# B&R Automation Studio project ASCommon
Automation Studio 6.5.0.306; technology packages: mappCockpit 6.6.0, mappMotion 6.6.1, mappSafety 6.4.1, mappServices 6.6.0, mappView 6.6.0, OpcUaCs 6.6.0

## Configuration X20CP1686X

CPU 5APC4100.TGL1-000, AutomationRuntime 6.5.1, Build 11.3.0, Vc 6.5.0

### Task classes (Cpu.sw)
```
Cyclic#1:
  MoveAxis <- Motion.MoveAxis.prg
  SimConnect <- SimConnect.prg
  BoxCreate <- BoxLift.BoxCreate.BoxCreate.prg [disabled]
  InfeedUp <- BoxLift.InfeedUp.InfeedUp.prg [disabled]
  InfeedLow <- BoxLift.InfeedLow.InfeedLow.prg [disabled]
  Lift <- BoxLift.Lift.Lift.prg [disabled]
  Unload <- BoxLift.Unload.Unload.prg [disabled]
  MachineMan <- BoxLift.MachineManager.MachineManager.prg [disabled]
  MachineMa1 <- BoxLiftOOP.MachineManager.prg
Cyclic#4:
  LampTest <- LampTest.prg
  RecipeMan <- Recipe.RecipeMan.prg
  SafetyCtrl <- Safety.SafetyCtrl.prg
DataObjects: McAcpSys
NcDataObjects: McDriveLog
Binaries: McAcpDrv, udbdef, McAcpSim, mvLoader, TCLang, TCData, FWRules, ArSvcReg, mvConfig, BRRole, sysconf, iomap, asfw, ashwac, UaCsConfig, Config_2, Config_1, ashwd, arconfig, Role, WebServ, User, TC, OpcUaCfg
Libraries: runtime, sys_lib, FileIO, AsZip, McBase, MpBase, MpAxis, McAcpAx, McAxis, SfDomain, MpCom, MpRecipe, CoTrace, AsTCP, AsIecCon, AsIODiag, UaCoal, SfDomVis, astime, standard, AsEPL, AsIOAcc, SfDomDrv, AsUSB, MpSfDomMgr, UaCoalPrv, ArUser, ArSsl, powerlnk, UaCore, AsIoTrc
```

### Hardware
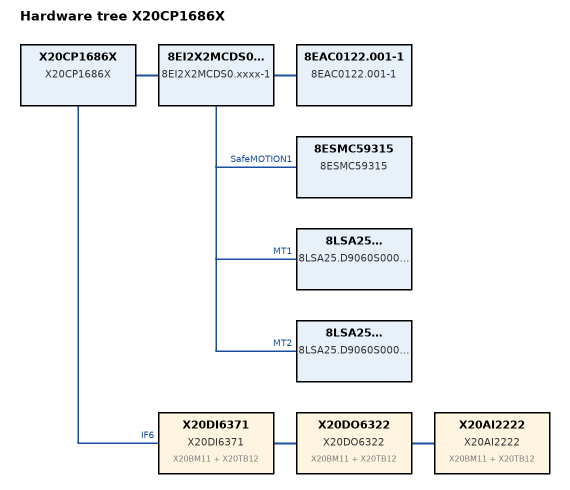
```
8EAC0122.001-1 : 8EAC0122.001-1 v3.0.0.0  [SS -> 8EI2X2MCDS0.xxxx-1.SS1]
  PlugInType = Encoder
  McAcoposTypeID = AcoposP3PlugInSConfig
  InterfaceType = Resolver
8EI2X2MCDS0.xxxx-1 : 8EI2X2MCDS0.xxxx-1 v2.4.0.3 (NodeNumber=1)  [PLK1 -> X20CP1686X.IF3 [Cable Type=PowerlinkCable, Length=10, Version=1.0.0.3]; MT2 -> 8LSA25.D9060S000-3a.MT]
  DriveConfiguration/Module:
    McAcoposTypeID = AcoposP3DConfig
    ActivateACOPOSSimulationOnPLC = 0
    PowerSupply = AC
  DriveConfiguration/Encoder:
    SafeEncInterface = EnDat22_SafeMOTION
  DriveConfiguration/Encoder/EncoderX41:
    InterfaceType = EnDatSafeMotion
  DriveConfiguration/Encoder/EncoderX42:
    InterfaceType = EnDatSafeMotion
  DriveConfiguration/Channel[1]/RealAxis:
    AxisReference = gAxis01
    MechanicalElementsIsInvisible = 0
  DriveConfiguration/Channel[1]/RealAxis/MechanicalElements/Gearbox:
    InputIsReadOnly = 0
    Input = 1
    OutputIsReadOnly = 0
    Output = 1
  DriveConfiguration/Channel[1]/RealAxis/MechanicalElements/RotaryToLinearTransformation:
    ReferenceDistanceIsReadOnly = 0
    ReferenceDistance = 1
  DriveConfiguration/Channel[1]/RealAxis:
    EncoderLink = OneEncoder
  DriveConfiguration/Channel[1]/RealAxis/Controller:
    ModeIsReadOnly = 0
    Mode = PositionController
  DriveConfiguration/Channel[1]/RealAxis/Homing:
    ModeIsReadOnly = 0
    Mode = Direct
    RestorePositionVariable = 
  DriveConfiguration/Channel[1]/RealAxis/StopReaction:
    QuickstopIsReadOnly = 0
    Quickstop = DecelerationLimit
    DriveErrorIsReadOnly = 0
    DriveError = DecelerationLimit
  DriveConfiguration/Channel[1]/RealAxis/MovementErrorLimits:
    PositionError = 10.0
    VelocityErrorMonitoring = Automatic1
  DriveConfiguration/Channel[1]/RealAxis:
    JerkFilterIsReadOnly = 0
    JerkFilter = NotUsed
    ZeroVibrationFilter = NotUsed
  DriveConfiguration/Channel[1]/RealAxis/DigitalInputs/HomingSwitch:
    SourceIsReadOnly = 0
    Source = NotUsed
    Level = High
  DriveConfiguration/Channel[1]/RealAxis/DigitalInputs/PositiveLimitSwitch:
    SourceIsReadOnly = 0
    Source = NotUsed
    Level = High
  DriveConfiguration/Channel[1]/RealAxis/DigitalInputs/NegativeLimitSwitch:
    SourceIsReadOnly = 0
    Source = NotUsed
    Level = High
  DriveConfiguration/Channel[1]/RealAxis/DigitalInputs/Trigger1:
    Source = X8Trigger1
    Level = High
  DriveConfiguration/Channel[1]/RealAxis/DigitalInputs/Trigger2:
    Source = X8Trigger2
    Level = High
  DriveConfiguration/Channel[1]/RealAxis/DigitalInputs/Quickstop:
    Input = Trigger2
  DriveConfiguration/Channel[1]/RealAxis/Simulation:
    SimulationModeOnPLC = SetValueGeneration
    SimulationModeOnACOPOS = NotUsed
  DriveConfiguration/Channel[1]:
    VirtualAxis = NotUsed
    ExternalEncoderAxis = NotUsed
  DriveConfiguration/Channel[2]/RealAxis:
    AxisReference = 
    MechanicalElementsIsInvisible = 0
  DriveConfiguration/Channel[2]/RealAxis/MechanicalElements/Gearbox:
    InputIsReadOnly = 0
    Input = 1
    OutputIsReadOnly = 0
    Output = 1
  DriveConfiguration/Channel[2]/RealAxis/MechanicalElements/RotaryToLinearTransformation:
    ReferenceDistanceIsReadOnly = 0
    ReferenceDistance = 1
  DriveConfiguration/Channel[2]/RealAxis:
    EncoderLink = OneEncoder
  DriveConfiguration/Channel[2]/RealAxis/Controller:
    ModeIsReadOnly = 0
    Mode = PositionController
  DriveConfiguration/Channel[2]/RealAxis/Homing:
    ModeIsReadOnly = 0
    Mode = Direct
    RestorePositionVariable = 
  DriveConfiguration/Channel[2]/RealAxis/StopReaction:
    QuickstopIsReadOnly = 0
    Quickstop = DecelerationLimit
    DriveErrorIsReadOnly = 0
    DriveError = DecelerationLimit
  DriveConfiguration/Channel[2]/RealAxis/MovementErrorLimits:
    PositionError = 10.0
    VelocityErrorMonitoring = Automatic1
  DriveConfiguration/Channel[2]/RealAxis:
    JerkFilterIsReadOnly = 0
    JerkFilter = NotUsed
    ZeroVibrationFilter = NotUsed
  DriveConfiguration/Channel[2]/RealAxis/DigitalInputs/HomingSwitch:
    SourceIsReadOnly = 0
    Source = NotUsed
    Level = High
  DriveConfiguration/Channel[2]/RealAxis/DigitalInputs/PositiveLimitSwitch:
    SourceIsReadOnly = 0
    Source = NotUsed
    Level = High
  DriveConfiguration/Channel[2]/RealAxis/DigitalInputs/NegativeLimitSwitch:
    SourceIsReadOnly = 0
    Source = NotUsed
    Level = High
  DriveConfiguration/Channel[2]/RealAxis/DigitalInputs/Trigger1:
    Source = X8Trigger1
    Level = High
  DriveConfiguration/Channel[2]/RealAxis/DigitalInputs/Trigger2:
    Source = X8Trigger2
    Level = High
  DriveConfiguration/Channel[2]/RealAxis/DigitalInputs/Quickstop:
    Input = Trigger2
  DriveConfiguration/Channel[2]/RealAxis/Simulation:
    SimulationModeOnPLC = SetValueGeneration
    SimulationModeOnACOPOS = NotUsed
  DriveConfiguration/Channel[2]:
    VirtualAxis = NotUsed
    ExternalEncoderAxis = NotUsed
8ESMC59315 : 8ESMC59315 v2.4.0.0  [SafeMOTION -> 8EI2X2MCDS0.xxxx-1.SafeMOTION1]
8LSA25.D9060S000-3 : 8LSA25.D9060S000-3 v2.2.0.2  [MT -> 8EI2X2MCDS0.xxxx-1.MT1]
  M1/MotorParameters:
    MOTOR_AMB_TEMP_RATED = 40
  M1/MotorParameters/TemperatureSensor:
    MOTOR_TEMPSENS_LIM = 130
8LSA25.D9060S000-3a : 8LSA25.D9060S000-3 v2.2.0.2  [MT -> 8EI2X2MCDS0.xxxx-1.MT2]
  M1/MotorParameters:
    MOTOR_AMB_TEMP_RATED = 40
  M1/MotorParameters/TemperatureSensor:
    MOTOR_TEMPSENS_LIM = 130
X20AI2222 : X20AI2222 v1.4.0.0  [SS1 -> X20TB12b.SS; SL -> X20BM11b.SL1]
X20BM11 : X20BM11 v1.1.0.0  [X2X1 -> X20CP1686X.IF6]
X20BM11a : X20BM11 v1.1.0.0  [X2X1 -> X20BM11.X2X2]
X20BM11b : X20BM11 v1.1.0.0  [X2X1 -> X20BM11a.X2X2]
X20CP1686X : X20CP1686X v1.8.2.0
  Connector IF2:
    ActivateDevice = 1
    HostName = ascommon
    Mode = Manual
    InternetAddress = 192.168.0.10
    SubnetMask = 255.255.255.0
    ActivateSnmp = 2
  Connector IF3:
    EplHostName = ascommon
    HostName = ascommon
  ConfigurationID = ASCommon_X20CP1686X
  Simulation = 1
  EnableUsbRemoteInstall = 1
  FileDevice1
  FileDeviceName1 = USER
  FileDevicePath1 = USER_PATH
  TimeZone = 140
  ActivateDaylightSavingTime = 1
  ActivateSntp = 1
  SntpcServAddr1 = 10.43.10.23
  SntpcServAddr2 = 10.43.10.24
  EthernetHostName = ascommon
  ActivateWebServer = 1
  HttpsSslCfg = WebServConf
  ActivateSdm = 1
X20DI6371 : X20DI6371 v1.2.2.0  [SS1 -> X20TB12.SS; SL -> X20BM11.SL1]
X20DO6322 : X20DO6322 v1.4.1.0  [SS1 -> X20TB12a.SS; SL -> X20BM11a.SL1]
X20TB12 : X20TB12 v1.0.0.0
X20TB12a : X20TB12 v1.0.0.0
X20TB12b : X20TB12 v1.0.0.0
```

### IoMap.iom - X20CP1686X/IoMap.iom
```iecst
VAR_CONFIG
	::LampTest:diSwitch AT %IX."X20DI6371".DigitalInput01;
	::SafetyCtrl:di_Reset AT %IX."X20DI6371".DigitalInput03;
	::LampTest:doLamp AT %QX."X20DO6322".DigitalOutput01;
	::LampTest:doLamp AT %QX."X20DO6322".DigitalOutput02;
	::LampTest:doLamp AT %QX."X20DO6322".DigitalOutput03;
END_VAR
```

### PvMap.vvm - X20CP1686X/PvMap.vvm
```iecst
VAR_CONFIG
	::InfeedUp:IO.doInfeed1Conveyor AT %Q.::SimConnect:SimOutputs.doInfeed1Conveyor; (*Insert your comment here...*)
	::InfeedUp:IO.aoInfeed1ConveyorSetSpeed AT %Q.::SimConnect:SimOutputs.aoInfeed1ConveyorSetSpeed; (*Insert your comment here...*)
	::SimConnect:SimInputs.diInfeed1BoxDetection AT %Q.::InfeedUp:IO.diInfeed1BoxDetection; (*Insert your comment here...*)
	::InfeedLow:IO.doInfeed2Conveyor AT %Q.::SimConnect:SimOutputs.doInfeed2Conveyor; (*Insert your comment here...*)
	::InfeedLow:IO.aoInfeed2ConveyorSetSpeed AT %Q.::SimConnect:SimOutputs.aoInfeed2ConveyorSetSpeed; (*Insert your comment here...*)
	::SimConnect:SimInputs.diInfeed2BoxDetection AT %Q.::InfeedLow:IO.diInfeed2BoxDetection; (*Insert your comment here...*)
	::BoxCreate:IO.aoEntrance1ConveyorSetSpeed AT %Q.::SimConnect:SimOutputs.aoEntrance1ConveyorSetSpeed; (*Insert your comment here...*)
	::BoxCreate:IO.aoEntrance2ConveyorSetSpeed AT %Q.::SimConnect:SimOutputs.aoEntrance2ConveyorSetSpeed; (*Insert your comment here...*)
	::BoxCreate:IO.aoInfeed1BoxCreationInterval AT %Q.::SimConnect:SimOutputs.aoInfeed1BoxCreationInterval; (*Insert your comment here...*)
	::BoxCreate:IO.aoInfeed2BoxCreationInterval AT %Q.::SimConnect:SimOutputs.aoInfeed2BoxCreationInterval; (*Insert your comment here...*)
	::BoxCreate:IO.doStopBoxCreation AT %Q.::SimConnect:SimOutputs.doStopBoxCreation; (*Insert your comment here...*)
	::Lift:IO.doLiftUp AT %Q.::SimConnect:SimOutputs.doLiftUp; (*Insert your comment here...*)
	::Lift:IO.doLiftDown AT %Q.::SimConnect:SimOutputs.doLiftDown; (*Insert your comment here...*)
	::Lift:IO.doLiftConveyor AT %Q.::SimConnect:SimOutputs.doLiftConveyor; (*Insert your comment here...*)
	::Lift:IO.aoLiftSetSpeed AT %Q.::SimConnect:SimOutputs.aoLiftSetSpeed; (*Insert your comment here...*)
	::Lift:IO.aoLiftConveyorSetSpeed AT %Q.::SimConnect:SimOutputs.aoLiftConveyorSetSpeed; (*Insert your comment here...*)
	::SimConnect:SimInputs.diLiftPositionInfeed1 AT %Q.::Lift:IO.diLiftPositionInfeed1; (*Insert your comment here...*)
	::SimConnect:SimInputs.diLiftPositionInfeed2 AT %Q.::Lift:IO.diLiftPositionInfeed2; (*Insert your comment here...*)
	::SimConnect:SimInputs.diLiftPositionUnload AT %Q.::Lift:IO.diLiftPositionUnload; (*Insert your comment here...*)
	::SimConnect:SimInputs.diLiftBoxDetection AT %Q.::Lift:IO.diLiftBoxDetection; (*Insert your comment here...*)
	::Unload:IO.aoUnloadConveyorSetSpeed AT %Q.::SimConnect:SimOutputs.aoUnloadConveyorSetSpeed; (*Insert your comment here...*)
	::SimConnect:SimInputs.diUnloadBoxDetection AT %Q.::Unload:IO.diUnloadBoxDetection; (*Insert your comment here...*)
END_VAR
```

### Config_1.axis - X20CP1686X/mappMotion/Config_1.axis
```
Element gAxis01 (Type=axis)
  BaseType = RotaryPeriodic
  MovementLimits = Internal
  Alarms = None
```

### Config_2.mprecipexml - X20CP1686X/mappServices/Config_2.mprecipexml
```
Element gRecipeXml (Type=mprecipexml)
  mapp.Gen:
    Enable = TRUE
    EnableCockpit = TRUE
    TaskClass = 4
    Audit = TRUE
    Parent
  mapp.Recipe.Xml:
    AutoSave = Standard
    Encryption = FALSE
    PassPhrase
    AutoExtension = TRUE
    Signature = Disabled
  Alarms = MpAlarmX
    mapp.AlarmX.Core.Configuration:
      [0]:
        Name = SaveFailed
        Message = {$BR/mapp/MpRecipeXml/Alarms/SaveFailed}
        Code = 0
        Severity = 1
        Behavior = EdgeAlarm
          AutoReset = TRUE
          Acknowledge = 1
          Confirm = 0
          MultipleInstances = TRUE
          ReactionWhilePending = TRUE
          Async = FALSE
          Recording:
            InactiveToActive = TRUE
            ActiveToInactive = FALSE
            UnacknowledgedToAcknowledged = TRUE
            UnconfirmedToConfirmed = TRUE
        Disable = FALSE
        AdditionalInformation1
        AdditionalInformation2
      [1]:
        Name = SaveFailedPartial
        Message = {$BR/mapp/MpRecipeXml/Alarms/SaveFailedPartial}
        Code = 0
        Severity = 1
        Behavior = EdgeAlarm
          AutoReset = TRUE
          Acknowledge = 1
          Confirm = 0
          MultipleInstances = TRUE
          ReactionWhilePending = TRUE
          Async = FALSE
          Recording:
            InactiveToActive = TRUE
            ActiveToInactive = FALSE
            UnacknowledgedToAcknowledged = TRUE
            UnconfirmedToConfirmed = TRUE
        Disable = FALSE
        AdditionalInformation1
        AdditionalInformation2
      [2]:
        Name = LoadFailed
        Message = {$BR/mapp/MpRecipeXml/Alarms/LoadFailed}
        Code = 0
        Severity = 1
        Behavior = EdgeAlarm
          AutoReset = TRUE
          Acknowledge = 1
          Confirm = 0
          MultipleInstances = TRUE
          ReactionWhilePending = TRUE
          Async = FALSE
          Recording:
            InactiveToActive = TRUE
            ActiveToInactive = FALSE
            UnacknowledgedToAcknowledged = TRUE
            UnconfirmedToConfirmed = TRUE
        Disable = FALSE
        AdditionalInformation1
        AdditionalInformation2
      [3]:
        Name = LoadFailedPartial
        Message = {$BR/mapp/MpRecipeXml/Alarms/LoadFailedPartial}
        Code = 0
        Severity = 1
        Behavior = EdgeAlarm
          AutoReset = TRUE
          Acknowledge = 1
          Confirm = 0
          MultipleInstances = TRUE
          ReactionWhilePending = TRUE
          Async = FALSE
          Recording:
            InactiveToActive = TRUE
            ActiveToInactive = FALSE
            UnacknowledgedToAcknowledged = TRUE
            UnconfirmedToConfirmed = TRUE
        Disable = FALSE
        AdditionalInformation1
        AdditionalInformation2
```

## Logical view

Binary libraries used (declarations not repeated): operator, runtime, astime, AsIecCon, brsystem, sys_lib, AsArSdm, AsZip, FileIO, standard, McBase 6.6.1, MpBase 6.6.0, MpAxis 6.6.1, McAcpAx 6.6.1, McAxis 6.6.1, SfDomain 6.4.1, MpCom 6.6.0, MpRecipe 6.6.0, CoTrace 6.6.0, MpAudit 6.6.0

### Password.txt
```
OPC UA Server:
	Nutzername: 	opcuauser
	Passwort:		.opcuauser

URL mappView Visu:
	http://127.0.0.1:81/index.html?visuId=mvStart
```

- Project.language (not shown)

### Global.var - Global variables
```iecst
VAR
	MpAxisParam : MpAxisBasicParType;
END_VAR
```


### Program Logical/Motion/MoveAxis (ANSIC)

#### Variables.var
```iecst
VAR
	Para : MpAxisBasicParType;
	mpAxisBasic_0 : MpAxisBasic;
END_VAR
```

#### compile_flags.txt
```
# This file is auto-generated by ASX. Do not edit manually, as changes may be overwritten.
# If you need to manually edit this file and prevent automatic updates, add "# MANUAL EDIT" to the first line.
-I
c:\projects_63\sps\Logical\Motion\MoveAxis
-I
c:\projects_63\sps\Temp\Includes\Motion\MoveAxis
-I
C:\Program Files (x86)\BrAutomation\AS6\AS\gnuinst\V11.3.0\6.0\i686-elf\include\c++\11.3.0
-I
C:\Program Files (x86)\BrAutomation\AS6\AS\gnuinst\V11.3.0\6.0\i686-elf\include\c++\11.3.0\i686-elf
-I
C:\Program Files (x86)\BrAutomation\AS6\AS\gnuinst\V11.3.0\6.0\i686-elf\include\c++\11.3.0\backward
-I
C:\Program Files (x86)\BrAutomation\AS6\AS\gnuinst\V11.3.0\6.0\lib\gcc\i686-elf\11.3.0\include
-I
C:\Program Files (x86)\BrAutomation\AS6\AS\gnuinst\V11.3.0\6.0\lib\gcc\i686-elf\11.3.0\include-fixed
-I
C:\Program Files (x86)\BrAutomation\AS6\AS\gnuinst\V11.3.0\6.0\i686-elf\include
-I
c:\projects_63\sps\Temp\Includes
-trigraphs
-fno-asm
-D
_DEFAULT_INCLUDES
-D
_SG4
--target=i686-elf
-fPIC
-Wall
```

#### Main.c
```c
#include <bur/plctypes.h>

#ifdef _DEFAULT_INCLUDES
	#include <AsDefault.h>
#endif

#define TRUE 1

void _INIT ProgramInit(void)
{
	mpAxisBasic_0.MpLink = &gAxis01;
	mpAxisBasic_0.Enable = TRUE;
	mpAxisBasic_0.Parameters = &Para;
}

void _CYCLIC ProgramCyclic(void)
{
	MpAxisBasic(&mpAxisBasic_0);
}

void _EXIT ProgramExit(void)
{

}
```

### Program Logical/Recipe/RecipeMan (IEC)

#### Cyclic.st - Cyclic code
```iecst
PROGRAM _INIT
	MpAxisParam := MpAxisParam;

	MpRecipeXml_0.Enable 	:= TRUE;
	MpRecipeXml_0.MpLink 	:= ADR(gRecipeXml);
	MpRecipeXml_0.DeviceName := ADR('Files');
	MpRecipeXml_0.FileName 	:= ADR(FileName);

	MpRecipeXml_0();

	MpRecipePar.Enable := TRUE;
	MpRecipePar.MpLink := ADR(gRecipeXml);
	MpRecipePar.PVName := ADR('MpAxisParam');

	MpRecipePar();

END_PROGRAM

PROGRAM _CYCLIC

	MpRecipeXml_0();
	MpRecipePar();

END_PROGRAM

PROGRAM _EXIT

	MpRecipeXml_0.Enable := FALSE;
	MpRecipeXml_0();

	MpRecipePar.Enable := FALSE;
	MpRecipePar();

END_PROGRAM
```

#### Variables.var - Local variables
```iecst
VAR
	MpRecipeXml_0 : MpRecipeXml;
	MpRecipePar : MpRecipeRegPar;
	FileName : {REDUND_UNREPLICABLE} STRING[80] := 'AxisParameter';
END_VAR
```

### Program Logical/Safety/SafetyCtrl (IEC)

#### Main.st - Init, cyclic, exit code
```iecst
PROGRAM _INIT

	MpAxisParam := MpAxisParam;
	gAxis01 	:= gAxis01;

END_PROGRAM

PROGRAM _CYCLIC

	di_Reset;

	diagCode_EStop;
	diagCode_LightCurtain;
	diagCode_Root;

END_PROGRAM

PROGRAM _EXIT

END_PROGRAM
```

#### Variables.var - Local variables
```iecst
VAR
	diagCode_EStop : UINT;
	diagCode_LightCurtain : UINT;
	diagCode_Root : UINT;
	di_Reset : BOOL;
END_VAR
```

### Package Logical/BoxLift - Project source code

### Package Logical/BoxLift/MachineManager - Automatic mode

### MachineManagerIF.typ - Module interface declaration (global visibility)
```iecst
TYPE
	AutomaticIFType : 	STRUCT  (*Communication interface for the Automatic module*)
		Cmd : AutomaticCmdType; (*Commands to the Automatic module*)
	END_STRUCT;
	AutomaticCmdType : 	STRUCT  (*Commands to the Automatic module*)
		Run : BOOL; (*Run the machine*)
	END_STRUCT;
END_TYPE
```

### MachineMangerIF.var - Module interface definition (global visibility)
```iecst
VAR
	gAutomatic : AutomaticIFType; (*Communication interface for the Automatic module*)
END_VAR
```

### Program Logical/BoxLift/MachineManager/MachineManager (IEC) - Automatic module functionality

#### Types.typ - Local data types
```iecst
(*Internal (private) data types*)

TYPE
	AutoStateEnum :
		(
		AUTO_IDLE,
		AUTO_WAIT_FOR_BOX,
		AUTO_PREPARE_UPPER_HANDOVER,
		AUTO_HANDOVER_UPPER_BOX,
		AUTO_PREPARE_LOWER_HANDOVER,
		AUTO_HANDOVER_LOWER_BOX,
		AUTO_HANDOVER_TO_UNLOAD,
		AUTO_UNLOAD_BOX
		);
END_TYPE
```

#### Variables.var - Local variables
```iecst
(*Internal (private) variables*)
VAR
	AutoState : AutoStateEnum;
	RunOld : BOOL; (*for edge detection of the Run command*)
END_VAR
```

#### MachineManager.st - Init, cyclic, exit code
```iecst
(*********************************************************************************
 * Copyright: B&R Industrial Automation GmbH
 * Author: B&R
 * Created: 2024-09-23
 * Description: Automatic control program
 *
 * The Automatic module controls the automatic machine sequence.
 *********************************************************************************)

PROGRAM _INIT

END_PROGRAM

PROGRAM _CYCLIC

	// Automatic mode switched off: reset all module commands and go to idle
	IF NOT gAutomatic.Cmd.Run AND RunOld THEN
		AutoState := AUTO_IDLE;
		gBoxCreate.Cmd.Run := FALSE;
		gInfeedUp.Cmd.Run := FALSE;
		gInfeedUp.Cmd.HandoverBox := FALSE;
		gInfeedLow.Cmd.Run := FALSE;
		gInfeedLow.Cmd.HandoverBox := FALSE;
		gLift.Cmd.HandoverBox := FALSE;
		gLift.Cmd.MoveBottom := FALSE;
		gLift.Cmd.MoveMiddle := FALSE;
		gLift.Cmd.MoveTop := FALSE;
		gLift.Cmd.ReceiveBox := FALSE;
		gUnload.Cmd.Run := FALSE;
	END_IF;

	RunOld := gAutomatic.Cmd.Run; // edge detection

	CASE AutoState OF
		AUTO_IDLE:
			// nothing to do

			// State transitions
			IF gAutomatic.Cmd.Run THEN
				AutoState := AUTO_WAIT_FOR_BOX;
			END_IF;

		//Create boxes and wait until a box has arrived at one of the infeeds
		AUTO_WAIT_FOR_BOX:
			gBoxCreate.Cmd.Run := TRUE;
			gInfeedUp.Cmd.Run := TRUE;
			gInfeedLow.Cmd.Run := TRUE;

			// State transitions
			IF gInfeedUp.Status.BoxAvailable THEN
				AutoState := AUTO_PREPARE_UPPER_HANDOVER;
				gBoxCreate.Cmd.Run := FALSE;
			ELSIF gInfeedLow.Status.BoxAvailable THEN
				AutoState := AUTO_PREPARE_LOWER_HANDOVER;
				gBoxCreate.Cmd.Run := FALSE;
			END_IF;

		//Move lift to the upper infeed position
		AUTO_PREPARE_UPPER_HANDOVER:
			gLift.Cmd.MoveTop := TRUE;

			// State transitions
			IF gLift.Status.InTopPosition THEN
				gLift.Cmd.MoveTop := FALSE;
				AutoState := AUTO_HANDOVER_UPPER_BOX;
			END_IF;

		//Handover a box from the upper infeed to the lift conveyor
		AUTO_HANDOVER_UPPER_BOX:
			gInfeedUp.Cmd.HandoverBox := TRUE;
			gLift.Cmd.ReceiveBox := TRUE;

			// State transitions
			IF gLift.Status.BoxDetected THEN
				gInfeedUp.Cmd.HandoverBox := FALSE;
				gInfeedUp.Cmd.Run := FALSE;
				gLift.Cmd.ReceiveBox := FALSE;
				AutoState := AUTO_HANDOVER_TO_UNLOAD;
			END_IF;

		//Move lift to the lower infeed position
		AUTO_PREPARE_LOWER_HANDOVER:
			gLift.Cmd.MoveMiddle := TRUE;

			// State transitions
			IF gLift.Status.InMiddlePosition THEN
				gLift.Cmd.MoveMiddle := FALSE;
				AutoState := AUTO_HANDOVER_LOWER_BOX;
			END_IF;

		//Handover a box from the lower infeed to the lift conveyor
		AUTO_HANDOVER_LOWER_BOX:
			gInfeedLow.Cmd.HandoverBox := TRUE;
			gLift.Cmd.ReceiveBox := TRUE;

			// State transitions
			IF gLift.Status.BoxDetected THEN
				gInfeedLow.Cmd.HandoverBox := FALSE;
				gInfeedLow.Cmd.Run := FALSE;
				gLift.Cmd.ReceiveBox := FALSE;
				AutoState := AUTO_HANDOVER_TO_UNLOAD;
			END_IF;

		//Handover a box from the lift to the unload conveyor
		AUTO_HANDOVER_TO_UNLOAD:
			gLift.Cmd.MoveBottom := TRUE;
			gUnload.Cmd.Run := TRUE;

			// State transitions
			IF EDGEPOS(gLift.Status.InBottomPosition) THEN
				gLift.Cmd.MoveBottom := FALSE;
				gLift.Cmd.HandoverBox := TRUE;
				// keep lift conveyor running for smooth handover
				AutoState := AUTO_UNLOAD_BOX;
			END_IF;

		// Keep running both lift and unload conveyors until box moved past unload sensor
		AUTO_UNLOAD_BOX:
			gUnload.Cmd.Run := TRUE;

			// State transitions
			IF EDGENEG(gUnload.Status.BoxDetected) THEN
				gLift.Cmd.HandoverBox := FALSE;
				gUnload.Cmd.Run := FALSE;
				AutoState := AUTO_WAIT_FOR_BOX;
			END_IF;

	END_CASE;

END_PROGRAM

PROGRAM _EXIT

END_PROGRAM
```

### Package Logical/BoxLift/BoxCreate - Box creation module

### BoxCreateIF.typ - Module interface declaration (global visibility)
```iecst
TYPE
	BoxCreateIFType : 	STRUCT  (*Communication interface for the Box Creation module*)
		Cmd : BoxCreateCmdType; (*Commands to the Box Creation module*)
		Par : BoxCreateParType; (*Parameters of the Box Creation module*)
	END_STRUCT;
	BoxCreateCmdType : 	STRUCT  (*Commands to the Box Creation module*)
		Run : BOOL; (*Create boxes at parametrized rates*)
	END_STRUCT;
	BoxCreateParType : 	STRUCT  (*Parameters of the Box Creation module*)
		UpperBoxCreationInterval : REAL := 20; (*Upper box creation interval*)
		UpperConveyorSpeed : REAL := 0.2; (*Set speed for the upper conveyor belt; unit [m/sec]*)
		LowerBoxCreationInterval : REAL := 25; (*Lower box creation interval*)
		LowerConveyorSpeed : REAL := 0.2; (*Set speed for the lower conveyor belt; unit [m/sec]*)
	END_STRUCT;
END_TYPE
```

### BoxCreateIF.var - Module interface definition (global visibility)
```iecst
VAR
	gBoxCreate : BoxCreateIFType; (*Communication interface for the Box Creation module*)
END_VAR
```

### Program Logical/BoxLift/BoxCreate/BoxCreate (IEC) - Box Creation module functionality

#### Types.typ - Local data types
```iecst
(*Internal (private) data types*)

TYPE
	IOType : 	STRUCT  (*Box Creation module IOs*)
		doStopBoxCreation : BOOL;
		aoInfeed1BoxCreationInterval : REAL := 20;
		aoInfeed2BoxCreationInterval : REAL := 25;
		aoEntrance1ConveyorSetSpeed : REAL;
		aoEntrance2ConveyorSetSpeed : REAL;
	END_STRUCT;
END_TYPE
```

#### Variables.var - Local variables
```iecst
(*Internal (private) variables*)
VAR
	IO : IOType; (*Box Creation module IOs*)
END_VAR
```

#### BoxCreate.st - Init, cyclic, exit code
```iecst
(*********************************************************************************
 * Copyright: B&R Industrial Automation GmbH
 * Author: B&R
 * Created: 2024-09-23
 * Description: Box Creation control program
 *
 * The Box Creation module generates boxes based on parametrized rates.
 *********************************************************************************)

PROGRAM _INIT

END_PROGRAM

PROGRAM _CYCLIC

	IF gBoxCreate.Cmd.Run THEN
		IO.doStopBoxCreation := FALSE;
		IO.aoInfeed1BoxCreationInterval := gBoxCreate.Par.UpperBoxCreationInterval;
		IO.aoInfeed2BoxCreationInterval := gBoxCreate.Par.LowerBoxCreationInterval;
		IO.aoEntrance1ConveyorSetSpeed := gBoxCreate.Par.UpperConveyorSpeed;
		IO.aoEntrance2ConveyorSetSpeed := gBoxCreate.Par.LowerConveyorSpeed;
	ELSE
		IO.doStopBoxCreation := TRUE;
		IO.aoInfeed1BoxCreationInterval := gBoxCreate.Par.UpperBoxCreationInterval;
		IO.aoInfeed2BoxCreationInterval := gBoxCreate.Par.LowerBoxCreationInterval;
		(*IO.aoEntrance1ConveyorSetSpeed := 0.0;
		IO.aoEntrance2ConveyorSetSpeed := 0.0;*)
	END_IF;

END_PROGRAM

PROGRAM _EXIT

END_PROGRAM
```

### Package Logical/BoxLift/InfeedUp - Upper Infeed module

### InfeedUpIF.typ - Module interface declaration (global visibility)
```iecst
TYPE
	InfeedUpIFType : 	STRUCT  (*Communication interface for the Upper Infeed module*)
		Cmd : InfeedUpCmdType; (*Commands to the Upper Infeed module*)
		Par : InfeedUpParType; (*Parameters of the Upper Infeed module*)
		Status : InfeedUpStatusType; (*Status of the Upper Infeed module*)
	END_STRUCT;
	InfeedUpCmdType : 	STRUCT  (*Commands to the Upper Infeed module*)
		Run : BOOL; (*Transport boxes along 2 conveyors*)
		HandoverBox : BOOL; (*Hand over the box to the next module*)
	END_STRUCT;
	InfeedUpParType : 	STRUCT  (*Parameters of the Upper Infeed module*)
		ConveyorSpeed : REAL := 0.2; (*Set speed for the conveyor belt; unit [m/sec]*)
	END_STRUCT;
	InfeedUpStatusType : 	STRUCT  (*Status of the Upper Infeed module*)
		BoxAvailable : BOOL; (*Box is available for handover at the end of the conveyor*)
	END_STRUCT;
END_TYPE
```

### InfeedUpIF.var - Module interface definition (global visibility)
```iecst
VAR
	gInfeedUp : InfeedUpIFType; (*Communication interface for the Upper Infeed module*)
END_VAR
```

### Program Logical/BoxLift/InfeedUp/InfeedUp (IEC) - Upper Infeed module functionality

#### Types.typ - Local data types
```iecst
(*Internal (private) data types*)

TYPE
	IOType : 	STRUCT  (*Upper Infeed module IOs*)
		diInfeed1BoxDetection : BOOL;
		doInfeed1Conveyor : BOOL;
		aoInfeed1ConveyorSetSpeed : REAL;
	END_STRUCT;
END_TYPE
```

#### Variables.var - Local variables
```iecst
(*Internal (private) variables*)
VAR
	IO : IOType; (*Upper Infeed module IOs*)
END_VAR
```

#### InfeedUp.st - Init, cyclic, exit code
```iecst
(*********************************************************************************
 * Copyright: B&R Industrial Automation GmbH
 * Author: B&R
 * Created: 2024-09-23
 * Description: Upper Infeed control program
 *
 * The Upper Infeed module transports the created boxes to the lift.
 * Set the Run command to
 *********************************************************************************)

PROGRAM _INIT

END_PROGRAM

PROGRAM _CYCLIC

	IF gInfeedUp.Cmd.Run THEN
		IO.doInfeed1Conveyor := NOT IO.diInfeed1BoxDetection;
		IF gInfeedUp.Cmd.HandoverBox THEN
			IO.doInfeed1Conveyor := TRUE;
		END_IF;
		IO.aoInfeed1ConveyorSetSpeed := gInfeedUp.Par.ConveyorSpeed;
	ELSE
		IO.doInfeed1Conveyor := FALSE;
		IO.aoInfeed1ConveyorSetSpeed := 0.0;
	END_IF;

	gInfeedUp.Status.BoxAvailable := IO.diInfeed1BoxDetection;

END_PROGRAM

PROGRAM _EXIT

END_PROGRAM
```

### Package Logical/BoxLift/InfeedLow - Lower Infeed module

### InfeedLowIF.typ - Module interface declaration (global visibility)
```iecst
TYPE
	InfeedLowIFType : 	STRUCT  (*Communication interface for the Lower Infeed module*)
		Cmd : InfeedLowCmdType; (*Commands to the Lower Infeed module*)
		Par : InfeedLowParType; (*Parameters of the Lower Infeed module*)
		Status : InfeedLowStatusType; (*Status of the Lower Infeed module*)
	END_STRUCT;
	InfeedLowCmdType : 	STRUCT  (*Commands to the Lower Infeed module*)
		Run : BOOL; (*Transport boxes along 2 conveyors*)
		HandoverBox : BOOL; (*Hand over the box to the next module*)
	END_STRUCT;
	InfeedLowParType : 	STRUCT  (*Parameters of the Lower Infeed module*)
		ConveyorSpeed : REAL := 0.2; (*Set speed for the conveyor belt; unit [m/sec]*)
	END_STRUCT;
	InfeedLowStatusType : 	STRUCT  (*Status of the Lower Infeed module*)
		BoxAvailable : BOOL; (*Box is available for handover at the end of the conveyor*)
	END_STRUCT;
END_TYPE
```

### InfeedLowIF.var - Module interface definition (global visibility)
```iecst
VAR
	gInfeedLow : InfeedLowIFType; (*Communication interface for the Upper Infeed module*)
END_VAR
```

### Program Logical/BoxLift/InfeedLow/InfeedLow (IEC) - Lower Infeed module functionality

#### Types.typ - Local data types
```iecst
(*Internal (private) data types*)

TYPE
	IOType : 	STRUCT  (*Lower Infeed module IOs*)
		diInfeed2BoxDetection : BOOL;
		doInfeed2Conveyor : BOOL;
		aoInfeed2ConveyorSetSpeed : REAL;
	END_STRUCT;
END_TYPE
```

#### Variables.var - Local variables
```iecst
(*Internal (private) variables*)
VAR
	IO : IOType; (*Lower Infeed module IOs*)
END_VAR
```

#### InfeedLow.st - Init, cyclic, exit code
```iecst
(*********************************************************************************
 * Copyright: B&R Industrial Automation GmbH
 * Author: B&R
 * Created: 2024-09-23
 * Description: Lower Infeed control program
 *
 * The Lower Infeed module transports the created boxes to the lift.
 *********************************************************************************)

PROGRAM _INIT

END_PROGRAM

PROGRAM _CYCLIC

	IF gInfeedLow.Cmd.Run THEN
		IO.doInfeed2Conveyor := NOT IO.diInfeed2BoxDetection;
		IF gInfeedLow.Cmd.HandoverBox THEN
			IO.doInfeed2Conveyor := TRUE;
		END_IF;
		IO.aoInfeed2ConveyorSetSpeed := gInfeedLow.Par.ConveyorSpeed;
	ELSE
		IO.doInfeed2Conveyor := FALSE;
		IO.aoInfeed2ConveyorSetSpeed := 0.0;
	END_IF;

	gInfeedLow.Status.BoxAvailable := IO.diInfeed2BoxDetection;

END_PROGRAM

PROGRAM _EXIT

END_PROGRAM
```

### Package Logical/BoxLift/Lift - Lift module

### LiftIF.typ - Module interface declaration (global visibility)
```iecst
TYPE
	LiftIFType : 	STRUCT  (*Communication interface for the Lift module*)
		Cmd : LiftCmdType; (*Commands to the Lift module*)
		Par : LiftParType; (*Parameters of the Lift module*)
		Status : LiftStatusType; (*Status of the Lift module*)
	END_STRUCT;
	LiftCmdType : 	STRUCT  (*Commands to the Lift module*)
		MoveTop : BOOL; (*Move to top position*)
		MoveMiddle : BOOL; (*Move to middle position*)
		MoveBottom : BOOL; (*Move to bottom position*)
		ReceiveBox : BOOL; (*Receive a box (by moving conveyor belt)*)
		HandoverBox : BOOL; (*Move to bottom position and handover box to next conveyor*)
	END_STRUCT;
	LiftParType : 	STRUCT  (*Parameters of the Lift module*)
		ConveyorSpeed : REAL := 0.2; (*Set speed for the conveyor belt; unit [m/sec]*)
		LiftSpeed : REAL := 0.2; (*Set speed for the lift; unit [m/sec]*)
	END_STRUCT;
	LiftStatusType : 	STRUCT  (*Status of the Lift module*)
		InTopPosition : BOOL;
		InMiddlePosition : BOOL;
		InBottomPosition : BOOL;
		BoxDetected : BOOL; (*Box detected by photo sensor in the center of the lift conveyor*)
	END_STRUCT;
END_TYPE
```

### LiftIF.var - Module interface definition (global visibility)
```iecst
VAR
	gLift : LiftIFType; (*Communication interface for the Lift module*)
END_VAR
```

### Program Logical/BoxLift/Lift/Lift (IEC) - Lift module functionality

#### Types.typ - Local data types
```iecst
(*Internal (private) data types*)

TYPE
	IOType : 	STRUCT  (*Lift module IOs*)
		diLiftPositionInfeed1 : BOOL;
		diLiftPositionInfeed2 : BOOL;
		diLiftPositionUnload : BOOL;
		diLiftBoxDetection : BOOL;
		doLiftUp : BOOL;
		doLiftDown : BOOL;
		doLiftConveyor : BOOL;
		aoLiftSetSpeed : REAL;
		aoLiftConveyorSetSpeed : REAL;
	END_STRUCT;
END_TYPE
```

#### Variables.var - Local variables
```iecst
(*Internal (private) variables*)
VAR
	IO : IOType; (*Upper Infeed module IOs*)
	TryUpwards : BOOL; (*For moving to middle position can be unclear whether to move the lift up or down*)
END_VAR
```

#### Lift.st - Init, cyclic, exit code
```iecst
(*********************************************************************************
 * Copyright: B&R Industrial Automation GmbH
 * Author: B&R
 * Created: 2024-09-23
 * Description: Lift control program
 *
 * The Lift module picks up boxes and moves them to the bottom position.
 *********************************************************************************)

PROGRAM _INIT

END_PROGRAM

PROGRAM _CYCLIC

	// Move lift to top position
	IF gLift.Cmd.MoveTop THEN
		IO.doLiftUp := NOT IO.diLiftPositionInfeed1;
		IO.doLiftDown := FALSE;
		IO.aoLiftSetSpeed := gLift.Par.LiftSpeed;
		IO.aoLiftConveyorSetSpeed := 0.0;
		IO.doLiftConveyor := FALSE;
	// Move lift to middle position
	ELSIF gLift.Cmd.MoveMiddle THEN
		IF IO.diLiftPositionInfeed1 THEN
			TryUpwards := FALSE;
		ELSIF IO.diLiftPositionUnload THEN
			TryUpwards := TRUE;
		END_IF;
		IF TryUpwards THEN
			IO.doLiftUp := NOT IO.diLiftPositionInfeed2 AND NOT IO.diLiftPositionInfeed1;
			IO.doLiftDown := FALSE;
		ELSE
			IO.doLiftDown := NOT IO.diLiftPositionInfeed2 AND NOT IO.diLiftPositionUnload;
			IO.doLiftUp := FALSE;
		END_IF;
		IO.aoLiftSetSpeed := gLift.Par.LiftSpeed;
		IO.aoLiftConveyorSetSpeed := 0.0;
		IO.doLiftConveyor := FALSE;
	// Move lift to bottom position
	ELSIF gLift.Cmd.MoveBottom THEN
		IO.doLiftDown := TRUE;
		IO.doLiftUp := FALSE;
		IO.aoLiftSetSpeed := gLift.Par.LiftSpeed;
		IO.aoLiftConveyorSetSpeed := 0.0;
		IO.doLiftConveyor := FALSE;
	// Receive box from previous machine module (move conveyor and wait)
	ELSIF gLift.Cmd.ReceiveBox THEN
		IO.doLiftConveyor := NOT IO.diLiftBoxDetection;
		IO.aoLiftConveyorSetSpeed := gLift.Par.ConveyorSpeed;
		IO.aoLiftSetSpeed := 0.0;
		IO.doLiftUp := FALSE;
		IO.doLiftDown := FALSE;
	// Handover box to next machine module (move conveyor and lift)
	ELSIF gLift.Cmd.HandoverBox THEN
		IO.aoLiftConveyorSetSpeed := gLift.Par.ConveyorSpeed;
		IO.aoLiftSetSpeed := 0;
		IO.doLiftConveyor := TRUE;
		IO.doLiftDown := FALSE;
		// No command set
	ELSE
		IO.doLiftUp := FALSE;
		IO.doLiftDown := FALSE;
		IO.doLiftConveyor := FALSE;
		IO.aoLiftConveyorSetSpeed := 0.0;
		IO.aoLiftSetSpeed := 0.0;
	END_IF;

	gLift.Status.InTopPosition := IO.diLiftPositionInfeed1;
	gLift.Status.InMiddlePosition := IO.diLiftPositionInfeed2;
	gLift.Status.InBottomPosition := IO.diLiftPositionUnload;
	gLift.Status.BoxDetected := IO.diLiftBoxDetection;

END_PROGRAM

PROGRAM _EXIT

END_PROGRAM
```

### Package Logical/BoxLift/Unload - Unload module

### UnloadIF.typ - Module interface declaration (global visibility)
```iecst
TYPE
	UnloadIFType : 	STRUCT  (*Communication interface for the Unload module*)
		Cmd : UnloadCmdType; (*Commands to the Unload module*)
		Par : UnloadParType; (*Parameters of the Unload module*)
		Status : UnloadStatusType; (*Status of the Unload module*)
	END_STRUCT;
	UnloadCmdType : 	STRUCT  (*Commands to the Unload module*)
		Run : BOOL; (*Transport box on Unload conveyor*)
	END_STRUCT;
	UnloadParType : 	STRUCT  (*Parameters of the Unload module*)
		ConveyorSpeed : REAL := 0.2; (*Set speed for the conveyor belt; unit [m/sec]*)
	END_STRUCT;
	UnloadStatusType : 	STRUCT  (*Status of the Unload module*)
		BoxDetected : BOOL; (*Box detected on Unload conveyor*)
	END_STRUCT;
END_TYPE
```

### UnloadIF.var - Module interface definition (global visibility)
```iecst
VAR
	gUnload : UnloadIFType; (*Communication interface for the Unload module*)
END_VAR
```

### Program Logical/BoxLift/Unload/Unload (IEC) - Unload module functionality

#### Types.typ - Local data types
```iecst
(*Internal (private) data types*)

TYPE
	IOType : 	STRUCT  (*Unload module IOs*)
		diUnloadBoxDetection : BOOL;
		aoUnloadConveyorSetSpeed : REAL;
	END_STRUCT;
END_TYPE
```

#### Variables.var - Local variables
```iecst
(*Internal (private) variables*)
VAR
	IO : IOType; (*Upper Infeed module IOs*)
	BoxCounter : UDINT := 0; (*counter of transported boxes*)
END_VAR
```

#### Unload.st - Init, cyclic, exit code
```iecst
(*********************************************************************************
 * Copyright: B&R Industrial Automation GmbH
 * Author: B&R
 * Created: 2024-09-23
 * Description: Unload control program
 *
 * The Unload module transports boxes away until they disappear.
 *********************************************************************************)

PROGRAM _INIT

END_PROGRAM

PROGRAM _CYCLIC

	IF gUnload.Cmd.Run THEN

		IO.aoUnloadConveyorSetSpeed := gUnload.Par.ConveyorSpeed;
	ELSE
		IO.aoUnloadConveyorSetSpeed := 0.0;
	END_IF;

	gUnload.Status.BoxDetected := IO.diUnloadBoxDetection;

	IF EDGEPOS(IO.diUnloadBoxDetection) THEN
		BoxCounter := BoxCounter + 1;
	END_IF

END_PROGRAM

PROGRAM _EXIT

END_PROGRAM
```

### Package Logical/BoxLiftOOP - Project source code OOP

### Program Logical/BoxLiftOOP/MachineManager (IEC_OOP)

- BoxLiftSTOOP.stpp - Method implementation (not shown)

- BoxLiftSTOOP.fub - Fub implementation (not shown)

- MachineManager.stpp - Init, cyclic, exit code (not shown)

#### MachineManager.typ - Local data types
```iecst
(*Internal (private) data types*)

TYPE
	AutoStateEnum :
		(
		AUTO_IDLE,
		AUTO_WAIT_FOR_BOX,
		AUTO_PREPARE_UPPER_HANDOVER,
		AUTO_HANDOVER_UPPER_BOX,
		AUTO_PREPARE_LOWER_HANDOVER,
		AUTO_HANDOVER_LOWER_BOX,
		AUTO_HANDOVER_TO_UNLOAD,
		AUTO_UNLOAD_BOX
		);
END_TYPE
```

#### MachineManager.var - Local variables
```iecst
VAR
	BoxUpConveyor : BoxCreateConveyor;
	BoxDownConveyor : BoxCreateConveyor;
	InfeedUpConveyor : Conveyor;
	InfeedDownConveyor : Conveyor;
	UnloadConveyor : Conveyor;
	Lift : LiftConveyor;
	Run : BOOL;
	AutoState : AutoStateEnum;
	RunOld : BOOL; (*for edge detection of the Run command*)

	(*IO simulation*)
	diBoxAvailableUp:BOOL;
	diBoxAvailableDown:BOOL;
	diBoxAvailableLift:BOOL;
	diLiftUp:BOOL;
	diLiftDown:BOOL;
	diLiftUnload:BOOL;
	diBoxDetectedUndload:BOOL;
END_VAR
```

- Visualisation Logical/mappView (not shown)

### Program Logical/LampTest (IEC)

#### Cyclic.ld - Cyclic code
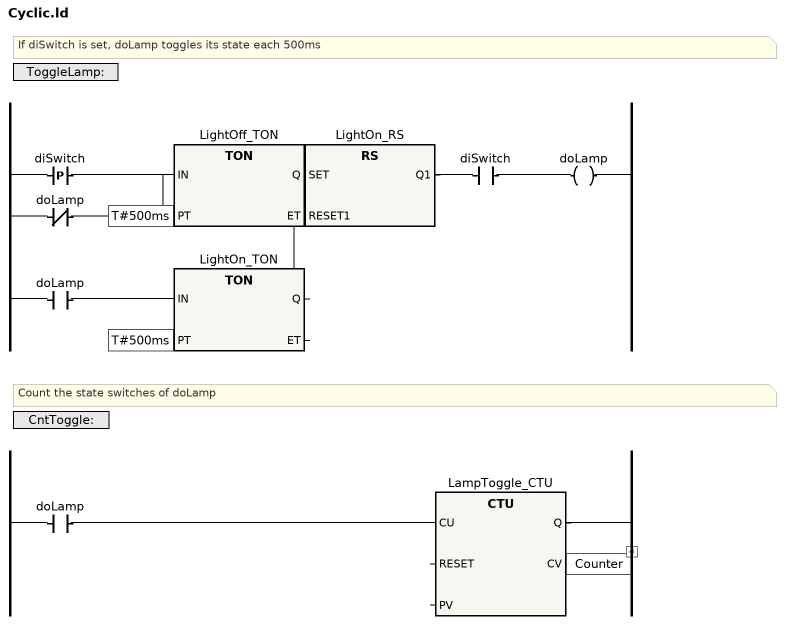
Diagram, in the editor's own instruction-list form stored in the file:
```il
PROGRAM _CYCLIC

VAR
	zz$$$$_0_r_trig_diSwitch : r_trig;
	zz$$$$_1_rf_trig_doLamp : rf_trig;
END_VAR

{NetworkNumber := 1}
(* If diSwitch is set, doLamp toggles its state each 500ms *)
ToggleLamp:
LD	diSwitch
ST	zz$$$$_0_r_trig_diSwitch.CLK
CAL	zz$$$$_0_r_trig_diSwitch
LD	zz$$$$_0_r_trig_diSwitch.Q
ORN	doLamp
ST	LightOff_TON.IN
LD	T#500ms
ST	LightOff_TON.PT
CAL	LightOff_TON
LD	doLamp
ST	LightOn_TON.IN
LD	T#500ms
ST	LightOn_TON.PT
CAL	LightOn_TON
LD	LightOff_TON.Q
ST	LightOn_RS.SET
LD	LightOn_TON.Q
ST	LightOn_RS.RESET1
CAL	LightOn_RS
LD	LightOn_RS.Q1
AND	diSwitch
ST	doLamp

{NetworkNumber := 2}
(* Count the state switches of doLamp *)
CntToggle:
LD	doLamp
ST	zz$$$$_1_rf_trig_doLamp.CLK
CAL	zz$$$$_1_rf_trig_doLamp
LD	zz$$$$_1_rf_trig_doLamp.Q
ST	LampToggle_CTU.CU
CAL	LampToggle_CTU
LD	LampToggle_CTU.CV
ST	Counter

END_PROGRAM
```

#### Variables.var - Local variables
```iecst
VAR
	doLamp : BOOL;
	diSwitch : BOOL;
	LightOn_RS : RS;
	LightOn_TON : TON;
	LightOff_TON : TON;
	Counter : UINT;
	LampToggle_CTU : CTU;
END_VAR
```

### Program Logical/SimConnect (IEC)

#### Types.typ
```iecst
TYPE
	SimOutputsType : 	STRUCT
		doLiftUp : BOOL; (*Move lift upwards*)
		doLiftDown : BOOL; (*Move lift downwards*)
		doInfeed1Conveyor : BOOL; (*Infeed1 Conveyor on/off*)
		doInfeed2Conveyor : BOOL; (*Infeed2e Conveyor on/off*)
		doLiftConveyor : BOOL; (*Lift conveyor on/off.*)
		doStopBoxCreation : BOOL := FALSE; (*Turns off/on creation of boxes*)
		aoInfeed1BoxCreationInterval : REAL := 20; (*Creation interval for boxes at top conveyor.*)
		aoInfeed2BoxCreationInterval : REAL := 25; (*Creation interval for boxes at bottom conveyor.*)
		aoEntrance1ConveyorSetSpeed : REAL := 0.6; (*Speed for ingoing conveyor top.*)
		aoEntrance2ConveyorSetSpeed : REAL := 0.5; (*Speed for ingoing bottom conveyor.*)
		aoInfeed1ConveyorSetSpeed : REAL := 0.7; (*Speed for outgoing top conveyor.*)
		aoInfeed2ConveyorSetSpeed : REAL := 0.7; (*Speed for outgoing bottom conveyor.*)
		aoLiftConveyorSetSpeed : REAL := 0.9; (*Speed for lift conveyor.*)
		aoLiftSetSpeed : REAL := 0.6; (*Travel speed between positions for the lift.*)
		aoUnloadConveyorSetSpeed : REAL := 0.9; (*Speed for unoad conveyor.*)
		doLiftPositionControl : BOOL; (*Switch from digital control (Up/Down) to position control of lift*)
		aoLiftPosition : REAL; (*Set position for lift in position control mode*)
	END_STRUCT;
	SimInputsType : 	STRUCT
		diLiftPositionInfeed1 : BOOL; (*Lift at position Infeed1 (top) *)
		diLiftPositionInfeed2 : BOOL; (*Lift at position Infeed2 (bottom) *)
		diLiftPositionUnload : BOOL := FALSE; (*Lift at unload position.*)
		diInfeed1BoxDetection : BOOL := FALSE; (*Box at infeed 1 conveyor unload position.*)
		diInfeed2BoxDetection : BOOL := FALSE; (*Box at bottom conveyor unload position.*)
		diLiftBoxDetection : BOOL := FALSE; (*Box loaded on lift.*)
		diUnloadBoxDetection : BOOL := FALSE; (*Box at unload conveyor.*)
	END_STRUCT;
END_TYPE
```

#### Variables.var
```iecst
VAR
	SimInputs : SimInputsType;
	SimOutputs : SimOutputsType := (aoLiftSetSpeed:=0.6);

	refactored : BOOL;

END_VAR
```

#### Main.st
```iecst
PROGRAM _INIT
	SimInputs;
	SimOutputs;
END_PROGRAM

PROGRAM _CYCLIC

	refactored;
	refactored;

END_PROGRAM

PROGRAM _EXIT

END_PROGRAM
```

Listed in the project but not available here: Logical/Global.typ, Logical/Recipe/RecipeMan/Types.typ, Logical/Safety/SafetyCtrl/Types.typ, Logical/LampTest/Types.typ
